# EPICS autosave request: TC/iocBoot/iocTC-IOC-01/tc_motor_extra.req
$(P)$(M)_AUTOONOFF_CMD
